PROGRAM MAIN
VAR
	ii, jj : INT;
END_VAR

END_PROGRAM

(* stored: Version 1.2.0.0, ProductVersion 3.1.4023.21
   POU MAIN: Id {2a06b1b8-2774-4e8b-aade-9ff87f2c5952}, SpecialFunc None *)
